(* PLC project SortingItemsByColour.project, CODESYS CODESYS V3.5 SP21 Patch 3 *)
(* stored: creationDateTime 2026-03-27T12:02:48.1085164, modificationDateTime 2026-03-27T12:01:55.6569734 *)

PROGRAM PLC_PRG
  VAR
    ItemLeftExitConveyor : R_TRIG;
    ItemEnteringExitConveyor : R_TRIG;
    ItemLeftEntryConveyor : F_TRIG;
    ExitConveyorStopped : F_TRIG;
    SceneStarted : R_TRIG;
    SwitchedToAutomatic : R_TRIG;
    GreenCount : WORD;
    BlueCount : WORD;
    MetalCount : WORD;
    ItemDetected : R_TRIG;
    ItemAtSensor : BOOL;
    StartPressed : R_TRIG;
    StopPressed : R_TRIG;
    ResetPressed : R_TRIG;
  END_VAR

                    ItemLeftExitConveyor(CLK:=FIO.iAtExit);
ItemEnteringExitConveyor(CLK:=FIO.iAtSensor);
ItemLeftEntryConveyor(CLK:=FIO.iAtSensor);
SceneStarted(CLK:= FIO.iRunning);
ItemAtSensor := FIO.iVisionSensor>0;
ItemDetected(CLK:=ItemAtSensor);
FIO.oGreen := GreenCount;
FIO.oBlue := BlueCount;
FIO.oMetal := MetalCount;
StartPressed(CLK:=FIO.iStart);
StopPressed(CLK:=FIO.iStop);
ResetPressed(CLK:=FIO.iReset);
FIO.oStartLight := FALSE;
FIO.oStopLight := FALSE;
FIO.oResetLight := FALSE;
ExitConveyorStopped(CLK:=FIO.oExitConveyor);
SwitchedToAutomatic(CLk:=FIO.iAutomatic);

IF SceneStarted.Q THEN
	FIO.oStackYellow := TRUE;
END_IF

IF SwitchedToAutomatic.Q THEN
	FIO.oEntryConveyor := TRUE;
	FIO.oStackGreen := TRUE;
END_IF

IF FIO.iManual THEN
	IF StartPressed.Q THEN
		FIO.oStartLight := TRUE;
		FIO.oEntryConveyor := TRUE;
		FIO.oStackGreen := TRUE;
	END_IF
END_IF

IF ItemEnteringExitConveyor.Q THEN
	FIO.oExitConveyor := TRUE;
END_IF

IF ItemLeftEntryConveyor.Q THEN
	FIO.oEntryConveyor := FALSE;
END_IF

IF ItemDetected.Q THEN
IF FIO.iVisionSensor >=1 AND FIO.iVisionSensor <=3 THEN
	FIO.oBlueSorterTurn := TRUE;
	FIO.oBlueSorterBelt := TRUE;
	FIO.oGreenSorterTurn := FALSE;
	FIO.oGreenSorterBelt := FALSE;
	FIO.oMetalSorterTurn := FALSE;
	FIO.oMetalSorterBelt := FALSE;
	BlueCount := BlueCount+1;

ELSIF FIO.iVisionSensor >=4 AND FIO.iVisionSensor <=6 THEN
	FIO.oGreenSorterTurn := TRUE;
	FIO.oGreenSorterBelt := TRUE;
	FIO.oBlueSorterTurn := FALSE;
	FIO.oBlueSorterBelt := FALSE;
	FIO.oMetalSorterTurn := FALSE;
	FIO.oMetalSorterBelt := FALSE;
	GreenCount := GreenCount+1;
	
ELSIF FIO.iVisionSensor >=7 AND FIO.iVisionSensor <=9 THEN
	FIO.oMetalSorterTurn := TRUE;
	FIO.oMetalSorterBelt := TRUE;
	FIO.oBlueSorterTurn := FALSE;
	FIO.oBlueSorterBelt := FALSE;
	FIO.oGreenSorterTurn := FALSE;
	FIO.oGreenSorterBelt := FALSE;
	MetalCount := MetalCount+1;
END_IF
END_IF

IF ItemLeftExitConveyor.Q THEN
	FIO.oExitConveyor := FALSE;
END_IF

IF ExitConveyorStopped.Q THEN
	FIO.oEntryConveyor := TRUE;
END_IF

IF FIO.iAtEnd THEN
	FIO.oBlueSorterTurn := FALSE;
	FIO.oBlueSorterBelt := FALSE;
	FIO.oGreenSorterTurn := FALSE;
	FIO.oGreenSorterBelt := FALSE;
	FIO.oMetalSorterTurn := FALSE;
	FIO.oMetalSorterBelt := FALSE;
	FIO.oEntryConveyor := FALSE;
	FIO.oExitConveyor := FALSE;
	FIO.oStackGreen := FALSE;
	FIO.oStackRed := TRUE;
END_IF

IF FIO.iManual THEN
IF StopPressed.Q THEN
	FIO.oBlueSorterBelt := FALSE;
	FIO.oGreenSorterBelt := FALSE;
	FIO.oMetalSorterBelt := FALSE;
	FIO.oEntryConveyor := FALSE;
	FIO.oExitConveyor := FALSE;
	FIO.oStackGreen := FALSE;
	FIO.oStackRed := FALSE;
	FIO.oStopLight := TRUE;
END_IF
END_IF

IF FIO.iManual THEN
IF ResetPressed.Q THEN
	FIO.oBlueSorterTurn := FALSE;
	FIO.oBlueSorterBelt := FALSE;
	FIO.oGreenSorterTurn := FALSE;
	FIO.oGreenSorterBelt := FALSE;
	FIO.oMetalSorterTurn := FALSE;
	FIO.oMetalSorterBelt := FALSE;
	FIO.oEntryConveyor := FALSE;
	FIO.oExitConveyor := FALSE;
	FIO.oStackGreen := FALSE;
	FIO.oStackRed := FALSE;
	FIO.oResetLight := TRUE;
END_IF
END_IF
                  
END_PROGRAM

CONFIGURATION Device
  RESOURCE Application ON PLC
    {attribute 'qualified_only'}
    VAR_GLOBAL  (* FIO *)
      iAtExit : BOOL;
      iAtSensor : BOOL;
      iVisionSensor : WORD;
      iRunning : BOOL;
      iAtEnd : BOOL;
      iAutomatic : BOOL;
      iManual : BOOL;
      iStart : BOOL;
      iStop : BOOL;
      iReset : BOOL;
      iEmergencyStop : BOOL;
      oEntryConveyor : BOOL;
      oExitConveyor : BOOL;
      oBlueSorterTurn : BOOL;
      oBlueSorterBelt : BOOL;
      oGreenSorterTurn : BOOL;
      oGreenSorterBelt : BOOL;
      oMetalSorterTurn : BOOL;
      oMetalSorterBelt : BOOL;
      oGreen : WORD;
      oBlue : WORD;
      oMetal : WORD;
      oStartLight : BOOL;
      oStopLight : BOOL;
      oResetLight : BOOL;
      oStackRed : BOOL;
      oStackYellow : BOOL;
      oStackGreen : BOOL;
    END_VAR
    TASK MainTask(INTERVAL := T#20ms, PRIORITY := 1);
    PROGRAM PLC_PRG WITH MainTask : PLC_PRG;
  END_RESOURCE
END_CONFIGURATION

CONFIGURATION Ethernet
END_CONFIGURATION

CONFIGURATION ModbusTCP_Server_Device
END_CONFIGURATION
